// TIA Portal V20 export
TYPE "FLink_Data"
// stored: IsFailsafeCompliant true, Namespace Safety
   STRUCT
      Word1 : Word;
      Word2 : Word;
      Word3 : Word;
      Word4 : Word;
      Word5 : Word;
      Word6 : Word;
      Word7 : Word;
      Word8 : Word;
      Word9 : Word;
      Word10 : Word;
      Word11 : Word;
      Word12 : Word;
      Word13 : Word;
      Word14 : Word;
      Word15 : Word;
      Word16 : Word;
      Word17 : Word;
      Word18_19 : DInt;
      Word20_21 : DInt;
      Word22_23 : DInt;
      Word24_25 : DInt;
      Word26_27 : DInt;
      Word28 : Word;
      Word29 : Word;
      Word30 : Word;
      Word31 : Word;
      Word32 : Word;
      Word33 : Word;
      Word34 : Word;
      Word35 : Word;
      Word36 : Word;
      Word37 : Word;
      Word38 : Word;
      Word39 : Word;
      Word40 : Word;
      Word41 : Word;
      Word42 : Word;
      Word43 : Word;
      Word44 : Word;
      Word45 : Word;
      Word46 : Word;
      Word47 : Word;
      Word48 : Word;
      Word49 : Word;
      Word50 : Word;
   END_STRUCT;
END_TYPE
